FUNCTION_BLOCK FB_MotorManipulator
VAR_INPUT
    bEnable  : BOOL;
    bExecute : BOOL;
	rPosition : REAL;
	bRefSens : BOOL;
END_VAR

VAR_IN_OUT
    ax : AXIS_REF;
  
END_VAR

VAR_OUTPUT
    eStatus : State;
END_VAR

VAR
    fbPower : MC_Power;
    fbMoveAbsolute : MC_MoveAbsolute;
    fbHalt : MC_Halt;
	fbHome : MC_HOME;
	fbReset : MC_Reset;
	
    bAxPower : BOOL;
    bAxMove : BOOL;
	bAxReset : BOOL;
    bHalt : BOOL;
	bAxRef : BOOL;
	
	nVelocity 	   : REAL := 15;
		
	bManEndMin AT%I* : BOOL := TRUE;
	bManEndMax AT%I* : BOOL := TRUE;

	bManBreakZ	AT%Q* : BOOL := FALSE;
	
	bGripperClosed AT%Q* :  BOOL;
	
	eState_manipulator : State_Motor_Manipulator := State_Motor_Manipulator.OFF;

END_VAR

ax.ReadStatus();

fbPower(Axis := ax, Enable := bAxPower, Enable_Positive := TRUE, Enable_Negative := TRUE);

fbReset(Axis := ax, Execute := bAxReset);

fbMoveAbsolute(Axis := ax, Execute := bAxMove, Position := rPosition, Velocity := nVelocity);

fbHome(Axis := ax, Execute := bRefSens, HomingMode := MC_DefaultHoming, bCalibrationCam := TRUE);

fbHalt(Axis := ax, Execute := bHalt);



IF NOT bEnable THEN
    eState_manipulator := 0;
    eStatus := State.Off;
    bAxPower := FALSE;
    bAxMove := FALSE;
	bAxReset := FALSE;
    bHalt := TRUE;
ELSE
    CASE eState_manipulator OF
		State_Motor_Manipulator.OFF:
			eStatus := State.Off;
            bAxPower := FALSE;
            bAxMove := FALSE;
            bHalt := TRUE;
			bAxReset := FALSE;
			
			IF bEnable THEN
				eState_manipulator := State_Motor_Manipulator.reset;
			END_IF
			
		State_Motor_Manipulator.reset:
			eStatus := State.init;
			bAxPower := FALSE;
			bAxMove := FALSE;
            bHalt := TRUE;
			bAxReset := TRUE;
			
			IF fbReset.Done THEN
				bAxReset := FALSE;
				eState_manipulator := State_Motor_Manipulator.init;
			END_IF
			
		State_Motor_Manipulator.init:
			bAxPower := TRUE;
			
			IF fbPower.Status AND bRefSens THEN
				eState_manipulator := State_Motor_Manipulator.REF;
			END_IF
			
		State_Motor_Manipulator.REF:
			bAxRef := TRUE;
			
			IF fbHome.Done THEN
				eState_manipulator := State_Motor_Manipulator.READY;
			END_IF
		
		State_Motor_Manipulator.READY:
			
			IF bExecute THEN
				eState_manipulator := State_Motor_Manipulator.PRODUCTION;
			END_IF
			
		State_Motor_Manipulator.PRODUCTION:
			bHalt := FALSE;
			bAxMove := TRUE;
			
			IF fbMoveAbsolute.Done THEN
				bAxMove := FALSE;
				bHalt := TRUE;
				eState_manipulator := State_Motor_Manipulator.READY;
			END_IF
			
			
			
			
	
	END_CASE
END_IF

END_FUNCTION_BLOCK

(* stored: Version 1.1.0.1, ProductVersion 3.1.4024.12
   POU FB_MotorManipulator: Id {69c0256a-531c-4ad4-b6bb-9ee8392ead5e}, SpecialFunc None *)
